// SIMATIC S7-200 project (STEP 7-Micro/WIN), CPU 226 REL 01.23

ORGANIZATION_BLOCK MAIN:OB1
TITLE=
// 项目信息：这个PLC程序控制K650吹瓶机。
// 物理设备包括K650吹瓶机、进料机构、加热区、吹瓶机构、冷却机构、出料机构、传感器和执行器。
// 
// 解析：
// 生产流程从启动按钮按下开始，系统启动后，进料阀门A和进料阀门B打开，将瓶胚送入设备。进料阀门只有在液位传感器未检测到满载、加热区温度传感器显示适宜温度、加热传感器和出料传感器正常、且无急停标志时才会动作，确保进料过程安全无溢料。进料完成后，加热器开始运行，将瓶胚加热至吹瓶所需温度。加热器只有在加热启用标志置位且加热区温度传感器确认温度达标时才会启动，保证瓶胚充分预热。随后，吹瓶机构将加热后的瓶胚吹制成瓶子，在系统确认加热流程结束后启动，避免因加热不足影响质量。
// 吹瓶完成后，冷却器启动，将成型瓶子冷却至适宜温度。冷却器在冷却启用标志置位时启动，确保瓶子冷却均匀、不变形。冷却结束后，出料阀门打开，将成品瓶送出生产线。出料阀门需在出料启用标志置位且出料传感器确认瓶子就位时才会动作，保证出料过程顺畅无堵塞。整个过程中，电机组驱动各环节，确保生产连续性。为保障安全，当急停按钮或急停信号触发时，系统暂停，所有设备停止运行，避免事故发生。
BEGIN
Network 1 // 网络标题
// 网络注释
LDN    V104.1
=      M1.1
?000
Network 2
LD     V600.5
JMP    3
Network 3
LD     I0.5
TON    T180, +2
Network 4
LD     V103.0
A      I3.2
A      I1.2
A      I0.6
A      I1.4
A      I1.1
AN     M1.1
AN     I3.0
AN     I3.1
AN     I3.5
AN     I3.4
AN     T180
LPS
=      M29.0
AN     M1.5
AN     I0.0
AN     M22.1
=      M1.4
LRD
LD     I0.0
O      M1.5
ALD
AN     M22.1
=      M1.5
LPP
LD     I2.5
O      M22.1
ALD
=      M22.1
Network 5
LD     M29.0
CALL   SBR_8:SBR8
Network 6
LD     M29.0
=      Q0.0
Network 7
LD     I0.4
TON    T181, +2
Network 8
LD     V103.0
A      I3.3
A      I0.6
A      I1.4
A      I1.1
AN     M1.1
AN     I3.0
AN     I3.1
AN     I3.5
AN     I3.4
AN     T181
LPS
=      M29.1
AN     M1.7
AN     I0.1
AN     M22.0
=      M1.6
LRD
LD     I0.1
O      M1.7
ALD
AN     M22.0
=      M1.7
LPP
LD     I2.6
O      M22.0
ALD
=      M22.0
Network 9
LD     M29.1
CALL   SBR_1:SBR1
Network 10
LD     M29.1
=      Q0.1
Network 11
LD     V103.0
A      I3.0
A      I1.4
AN     M1.1
AN     I3.2
AN     I3.3
AN     I3.5
AN     I3.4
LDN    I0.7
O      M29.2
ALD
LPS
AN     T214
=      M29.2
LRD
AN     M29.3
AN     M15.1
=      M2.1
LRD
AN     M2.1
TON    T34, +50
LRD
LD     M2.1
O      Q2.2
ALD
AN     T34
AN     M15.1
=      Q2.2
LRD
LD     I2.1
O      M29.3
ALD
AN     M15.1
=      M29.3
LPP
LD     I0.7
O      M15.1
ALD
LPS
AN     T214
=      M15.1
LPP
TON    T214, +5
Network 12
LD     M29.2
CALL   SBR_2:SBR2
Network 13
LD     M29.2
AN     Q0.0
=      Q0.2
Network 14
LD     V103.0
A      I3.1
A      I1.4
AN     M1.1
AN     I3.2
AN     I3.3
AN     I3.5
AN     I0.6
AN     I3.4
LPS
=      M2.3
A      I0.7
AN     M15.3
AN     M15.4
=      M15.2
LRD
AN     I0.7
AN     M15.4
AN     M24.5
=      M15.3
LPP
LD     M24.5
O      M15.4
ALD
=      M15.4
Network 15
LD     M2.3
CALL   SBR_2:SBR2
Network 16
LD     M2.3
=      Q0.3
Network 17
LD     V103.0
A      I3.5
A      I1.4
AN     M1.1
AN     I3.2
AN     I3.3
AN     I3.1
AN     I3.0
AN     I1.0
LPS
=      M29.4
AN     M29.5
AN     I2.3
=      M2.5
LPP
LD     I2.3
O      M29.5
ALD
=      M29.5
Network 18
LD     M29.4
CALL   SBR_3:SBR3
Network 19
LD     M29.4
=      Q1.0
Network 20
LD     V103.0
A      I3.4
A      I1.4
AN     M1.1
AN     I3.2
AN     I3.3
AN     I3.0
AN     I3.1
AN     I1.1
=      M2.7
MOVW   VW452, VW180
MOVW   VW454, VW182
Network 21
LD     M2.7
=      Q1.1
Network 22
LD     V103.0
A      V101.5
A      I1.4
AN     M1.1
=      Q1.2
Network 23
LD     V101.4
A      I1.4
AN     M1.1
=      Q1.3
Network 24
LD     I1.3
TON    T182, +2
Network 25
LD     I3.2
A      V103.1
A      I0.4
A      I1.5
A      I1.4
A      I2.0
AN     M1.1
AN     I3.0
AN     I3.1
AN     I3.4
AN     I3.5
AN     T182
LPS
=      M30.3
AN     M3.2
AN     I0.2
AN     M22.2
=      M3.1
LRD
LD     I0.2
O      M3.2
ALD
AN     M22.2
=      M3.2
LPP
LD     I2.7
O      M22.2
ALD
=      M22.2
Network 26
LD     M30.3
CALL   SBR_4:SBR4
Network 27
LD     M30.3
=      Q1.4
Network 28
LD     I1.2
TON    T183, +2
Network 29
LD     I3.3
A      V103.1
A      I1.5
A      I1.4
A      I2.0
AN     M1.1
AN     I3.0
AN     I3.1
AN     I3.4
AN     I3.5
AN     T183
LPS
=      M30.4
AN     M3.5
AN     I0.3
AN     M22.3
=      M3.4
LRD
LD     I0.3
O      M3.5
ALD
AN     M22.3
=      M3.5
LPP
LD     I3.6
O      M22.3
ALD
=      M22.3
Network 30
LD     M30.4
CALL   SBR_5:SBR5
Network 31
LD     M30.4
=      Q1.5
Network 32
LD     I3.0
A      V103.1
A      I1.4
AN     M1.1
AN     I3.2
AN     I3.3
AN     I3.5
AN     I3.4
LDN    I1.6
O      M29.6
ALD
LPS
AN     T213
=      M29.6
LRD
AN     M29.7
AN     M15.0
=      M3.7
LRD
AN     M3.7
TON    T35, +50
LRD
LD     M3.7
O      Q2.3
ALD
AN     T35
AN     M15.0
=      Q2.3
LRD
LD     I2.2
O      M29.7
ALD
AN     M15.0
=      M29.7
LPP
LD     I1.6
O      M15.0
ALD
LPS
AN     T213
=      M15.0
LPP
TON    T213, +5
Network 33
LD     M29.6
CALL   SBR_2:SBR2
Network 34
LD     M29.6
AN     Q1.4
=      Q1.6
Network 35
LD     I3.1
A      V103.1
A      I1.4
AN     M1.1
AN     I3.2
AN     I3.3
AN     I3.4
AN     I1.5
AN     I3.5
LPS
=      M4.1
A      I1.6
AN     M15.7
AN     M15.6
=      M15.5
LRD
AN     I1.6
AN     M15.7
AN     M24.5
=      M15.6
LPP
LD     M24.5
O      M15.7
ALD
=      M15.7
Network 36
LD     M4.1
CALL   SBR_2:SBR2
Network 37
LD     M4.1
=      Q2.0
Network 38
LD     I3.5
A      V103.1
A      I1.4
AN     M1.1
AN     I3.2
AN     I3.3
AN     I3.1
AN     I3.0
AN     I1.7
LPS
=      M30.0
AN     M30.1
AN     I2.4
=      M4.3
LPP
LD     I2.4
O      M30.1
ALD
=      M30.1
Network 39
LD     M30.0
CALL   SBR_3:SBR3
Network 40
LD     M30.0
=      Q0.4
Network 41
LD     I3.4
A      V103.1
A      I1.4
AN     M1.1
AN     I3.2
AN     I3.3
AN     I3.0
AN     I3.1
AN     I3.1
AN     I2.0
=      M4.5
MOVW   VW452, VW180
MOVW   VW454, VW182
Network 42
LD     M4.5
=      Q0.5
Network 43
LD     V101.5
A      V103.1
A      I1.4
AN     M1.1
=      Q0.6
Network 44
LD     M4.5
O      M4.3
O      M15.5
O      M15.6
O      M3.7
O      M3.4
O      M3.1
O      M2.7
O      M2.5
O      M15.3
O      M15.2
O      M1.6
O      M2.1
O      M1.4
=      Q1.7
Network 45
LD     M1.1
=      V600.5
Network 46
LD     V104.1
O      SM0.1
O      V100.2
R      M10.0, 8
R      M11.0, 2
R      M12.0, 8
R      M13.0, 2
Network 47
LBL    3
Network 48
LDN    V600.5
JMP    1
Network 49
LD     M10.0
O      M10.1
O      M10.2
O      M10.3
=      M20.0
Network 50
LD     M12.0
O      M12.1
O      M12.2
O      M12.3
=      M20.1
Network 51
LDN    M5.6
ON     M5.1
A      M5.2
AN     V104.1
EU
=      M4.7
Network 52
LDN    M5.7
ON     M20.5
A      M5.3
AN     V104.1
EU
=      M5.0
Network 53
LD     M4.7
S      M5.1, 1
Network 54
LD     M5.0
S      M20.5, 1
Network 55
LD     M10.0
A      V100.6
S      M25.2, 1
Network 56
LD     M12.0
A      V100.5
S      M25.3, 1
Network 57
LD     V100.2
O      SM0.1
O      M17.7
LD     V100.3
O      V100.4
ED
OLD
R      M25.2, 2
Network 58
LD     V100.1
S      M7.0, 1
Network 59
LD     SM0.0
MOVW   VW204, VW3800
/I     +2, VW3800
MOVW   VW3800, VW3900
+I     +30, VW3900
Network 60
LD     M7.0
TON    T44, VW3900
Network 61
LD     M10.0
O      SM0.1
O      M27.0
R      M7.0, 1
Network 62
LD     V100.6
AN     M25.2
O      V100.4
AN     M20.1
LD     V100.6
O      V100.4
AN     V100.5
A      V100.1
LD     V100.6
A      V100.5
A      T44
OLD
ALD
LD     T97
A      M7.6
AN     M25.2
OLD
A      M1.1
=      M5.2
Network 63
LD     V100.5
AN     M25.3
O      V100.3
AN     M20.0
A      V100.1
LD     T99
A      M7.6
AN     M25.3
OLD
A      M1.1
=      M5.3
Network 64
LD     V100.1
R      V100.2, 1
Network 65
LD     M4.7
O      M5.0
R      V100.1, 1
Network 66
LD     V100.5
AN     V100.6
LD     V100.6
AN     V100.5
OLD
O      V100.4
O      V100.3
S      M6.0, 1
Network 67
LDN    V100.6
AN     V100.5
O      M20.3
R      M6.2, 1
R      M5.1, 1
R      M20.5, 1
A      Q0.6
A      Q1.2
R      M6.0, 1
Network 68
LDN    V100.6
ON     V100.5
A      M1.1
R      M6.1, 1
Network 69
LD     M5.6
A      M1.1
A      V100.5
TON    T99, VW1316
Network 70
LD     T99
S      V2100.0, 1
Network 71
LD     M12.0
R      V2100.0, 1
Network 72
LD     M12.0
O      V104.1
O      M20.4
O      V100.2
O      M27.0
R      M5.6, 1
Network 73
LD     M1.1
EU
=      M20.4
Network 74
LD     V100.5
A      M10.0
S      M5.6, 1
Network 75
LD     M5.7
A      M1.1
A      V100.6
TON    T97, VW1316
Network 76
LD     T97
S      V2100.1, 1
Network 77
LD     M10.0
R      V2100.1, 1
Network 78
LD     M10.0
O      V104.1
O      M20.3
O      V100.2
O      M27.0
R      M5.7, 1
Network 79
LD     M1.1
EU
=      M20.3
Network 80
LD     V100.6
A      M12.0
S      M5.7, 1
Network 81
LD     V100.6
A      V100.5
S      M6.1, 1
S      M6.2, 1
=      M7.6
Network 82
LD     V100.3
O      V100.2
R      M13.3, 1
Network 83
LD     V100.4
O      V100.2
R      M11.3, 1
Network 84
LDN    M6.5
=      M6.3
Network 85
LD     SM0.1
O      M11.1
O      V100.2
O      V104.1
O      M27.0
R      M6.3, 1
R      M6.5, 1
Network 86
LDN    V100.5
S      M25.0, 1
Network 87
LD     V100.5
A      M10.0
R      M25.0, 1
Network 88
LD     M4.7
A      I0.4
A      I1.2
A      M6.3
LD     M10.0
A      I1.3
OLD
LD     M10.1
A      T139
A      I1.6
OLD
LD     T49
O      T119
O      T120
A      M10.2
AN     V108.5
OLD
LD     M10.3
A      I1.2
LD     M10.4
A      T52
A      I1.7
OLD
LD     M10.5
A      T198
OLD
LD     M10.6
A      T53
OLD
LD     M10.7
A      T148
A      I1.7
OLD
LD     M11.0
A      I1.5
OLD
LD     V108.5
A      T178
OLD
OLD
LD     I2.0
O      T119
O      T120
A      V108.5
A      M10.2
A      T140
LD     M11.1
AN     V108.5
OLD
A      I2.0
OLD
EU
=      M6.4
Network 89
LD     M10.5
TON    T198, +1
Network 90
LD     M11.1
A      V108.5
TON    T178, +5
Network 91
LD     M10.2
A      V108.5
TON    T140, +1
Network 92
LD     M11.2
=      M20.6
Network 93
LD     M11.2
A      M20.7
AN     V100.2
AN     V100.4
LD     I2.0
AN     V108.5
O      V108.5
ALD
A      I1.2
LD     V2100.1
O      M25.0
ALD
LD     V100.6
A      V100.5
O      V100.6
ALD
O      M6.4
A      M1.1
EU
SHRB   M6.3, M10.0, +16
Network 94
LD     M20.6
=      M20.7
Network 95
LD     M10.0
TON    T47, VW950
Network 96
LD     I1.3
TON    T184, +2
Network 97
LD     M10.0
A      T47
LD     M31.5
AN     T184
OLD
A      I1.5
A      I1.4
A      I0.4
LD     I2.0
AN     V108.5
O      V108.5
ALD
A      M1.1
LPS
S      M6.5, 1
=      M31.5
LD     I1.2
O      M6.6
ALD
AN     M6.7
AN     M23.2
=      M6.6
LRD
LD     I0.2
O      M6.7
ALD
AN     M23.2
=      M6.7
LPP
LD     I2.7
O      M23.2
ALD
=      M23.2
Network 98
LD     M31.5
CALL   SBR_4:SBR4
Network 99
LDN    M31.5
TON    T48, VW952
Network 100
LD     M10.1
A      T48
A      I1.4
A      M1.1
A      I1.3
LPS
AN     T139
=      M30.5
LRD
LD     I1.5
O      M30.6
ALD
AN     M8.1
AN     M14.0
=      M30.6
LRD
AN     M30.6
TON    T35, +50
LRD
LD     M30.6
O      Q2.3
ALD
AN     T35
AN     M14.0
=      Q2.3
LRD
LD     I2.2
O      M8.1
ALD
AN     M14.0
=      M8.1
LPP
LD     I1.6
O      M14.0
ALD
LPS
AN     T139
=      M14.0
LPP
TON    T139, +2
Network 101
LD     M30.5
CALL   SBR_2:SBR2
Network 102
LDN    M30.5
TON    T109, VW908
Network 103
LD     M10.1
EU
S      V200.1, 1
Network 104
LD     T199
O      SM0.1
O      M27.0
R      V200.1, 1
Network 105
LD     V200.1
=      M19.6
TON    T100, VW62
Network 106
LD     M10.3
TON    T50, VW956
Network 107
LD     I1.2
TON    T185, +2
Network 108
LD     T50
A      M10.3
LD     M31.6
AN     T185
OLD
A      I2.0
A      I1.4
A      I1.6
A      M1.1
O      M27.5
LPS
=      M31.6
LD     I1.3
O      M27.5
O      M8.4
ALD
AN     M8.5
AN     M23.3
=      M8.4
LRD
LD     I0.3
O      M8.5
ALD
AN     M23.3
=      M8.5
LPP
LD     I3.6
O      M23.3
ALD
=      M23.3
Network 109
LD     M31.6
CALL   SBR_5:SBR5
Network 110
LDN    M31.6
TON    T51, VW958
Network 111
LD     M10.4
A      T51
O      M31.7
A      I1.4
A      M1.1
A      I1.2
LPS
AN     T133
=      M31.7
LRD
AN     M31.0
AN     I2.4
AN     M24.6
AN     I1.7
=      M8.7
LRD
LD     I2.4
O      M31.0
ALD
AN     I1.7
AN     M24.6
=      M31.0
LPP
A      I1.7
LPS
AN     T133
=      M24.6
LPP
TON    T133, VW978
Network 112
LD     M10.7
AN     I1.7
=      M26.3
Network 113
LD     M31.7
O      M26.3
CALL   SBR_3:SBR3
Network 114
LD     M10.4
TON    T166, VW960
Network 115
LD     M10.4
A      T166
A      M1.1
A      I1.4
=      Q0.6
TON    T52, VW204
Network 116
LD     M12.5
A      V100.5
A      V100.6
O      V100.6
O      V100.3
O      V100.5
O      V100.4
A      M1.1
A      M10.6
TON    T53, VW210
=      V600.1
Network 117
LD     M11.0
TON    T55, VW966
Network 118
LD     M10.7
TON    T148, +1
Network 119
LD     T55
A      M11.0
O      M27.3
AN     I1.5
LPS
A      M1.1
=      M9.1
LPP
LD     I1.6
ON     I1.6
ALD
=      M14.5
Network 120
LD     M9.1
CALL   SBR_2:SBR2
Network 121
LD     M9.1
A      M1.1
O      M27.3
AN     I1.5
LD     Q0.0
A      V100.5
AN     Q0.6
AN     V100.4
AN     V100.6
OLD
=      Q2.0
Network 122
LD     M11.1
TON    T58, VW964
Network 123
LD     V600.1
TON    T54, VW980
Network 124
LD     M11.1
A      T58
A      I1.4
AN     V108.5
A      I1.5
A      M1.1
LD     M10.2
A      V108.5
OLD
LDN    T54
A      V600.1
OLD
O      M27.4
AN     I2.0
=      M8.2
MOVW   VW452, VW180
MOVW   VW454, VW182
Network 125
LD     M8.2
O      M27.4
A      M1.1
=      Q0.5
Network 126
LDN    M9.6
A      M1.1
=      M9.2
Network 127
LD     SM0.1
O      M13.1
O      V100.2
O      V104.1
O      M17.7
R      M9.2, 1
R      M9.6, 1
Network 128
LDN    V100.6
S      M25.1, 1
Network 129
LD     V100.6
A      M12.0
R      M25.1, 1
Network 130
LD     M5.0
A      I1.2
A      I0.4
A      M9.2
LD     M12.0
A      I0.5
OLD
LD     M12.1
A      I0.7
A      T131
OLD
LD     T39
O      T119
O      T120
A      M12.2
AN     V108.5
OLD
LD     M12.3
A      I0.4
LD     M12.4
A      T42
A      I1.0
OLD
LD     M12.5
A      T159
OLD
LD     M12.6
A      T43
OLD
LD     M12.7
A      T149
A      I1.0
OLD
LD     M13.0
A      I0.6
OLD
LD     T143
A      V108.5
OLD
OLD
LD     I1.1
O      T39
O      T119
A      T141
A      M12.2
A      V108.5
LD     M13.1
AN     V108.5
OLD
A      I1.1
OLD
EU
=      M9.3
Network 131
LD     M13.1
A      V108.5
TON    T143, +5
Network 132
LD     M12.2
A      V108.5
TON    T141, +1
Network 133
LD     M12.5
TON    T159, +1
Network 134
LD     M12.7
TON    T149, +1
Network 135
LD     M13.2
=      M21.0
Network 136
LD     M13.2
A      M21.1
LD     V2100.0
O      M25.1
ALD
AN     V100.2
AN     V100.3
LD     I1.1
AN     V108.5
O      V108.5
ALD
A      I0.4
LD     V100.5
A      V100.6
O      V100.5
ALD
O      M9.3
A      M1.1
EU
SHRB   M9.2, M12.0, +16
Network 137
LD     M21.0
=      M21.1
Network 138
LD     M12.0
TON    T37, VW900
Network 139
LD     I0.5
TON    T186, +2
Network 140
LD     I1.1
AN     V108.5
O      V108.5
LD     M12.0
A      T37
LD     M28.0
AN     T186
OLD
ALD
A      I0.6
A      I1.4
A      M1.1
A      I1.2
LPS
=      M28.0
LD     I0.4
O      M9.4
ALD
AN     M9.5
AN     I0.0
AN     M23.0
=      M9.4
LRD
LD     I0.0
O      M9.5
ALD
AN     M23.0
=      M9.5
LRD
S      M9.6, 1
LPP
LD     I2.5
O      M23.0
ALD
=      M23.0
Network 141
LD     M28.0
CALL   SBR_8:SBR8
Network 142
LDN    M28.0
TON    T38, VW904
Network 143
LD     M12.1
A      T38
A      I1.4
A      M1.1
A      I0.5
LPS
AN     T131
=      M31.1
LRD
LD     I0.6
O      M31.2
ALD
AN     M17.0
AN     M14.1
=      M31.2
LRD
AN     M31.2
TON    T36, +50
LRD
LD     M31.2
O      Q2.2
ALD
AN     T36
AN     M14.1
=      Q2.2
LRD
LD     I2.1
O      M17.0
ALD
AN     M14.1
=      M17.0
LPP
LD     I0.7
O      M14.1
ALD
LPS
AN     T131
=      M14.1
LPP
TON    T131, +2
Network 144
LD     M31.1
CALL   SBR_2:SBR2
Network 145
LDN    M31.1
TON    T114, VW908
Network 146
LD     M12.1
EU
S      V200.0, 1
Network 147
LD     T199
O      M27.0
O      SM0.1
R      V200.0, 1
Network 148
LD     V200.0
=      M19.7
TON    T98, VW60
Network 149
LD     T98
O      T100
LD     Q2.1
AN     T199
OLD
=      Q2.1
Network 150
LD     Q2.1
TON    T199, VW236
Network 151
LD     M12.3
TON    T40, VW912
Network 152
LD     I0.4
TON    T187, +2
Network 153
LD     M12.3
A      T40
LD     M28.1
AN     T187
OLD
A      I1.1
A      I1.4
A      M1.1
A      I0.7
O      M27.2
LPS
=      M28.1
LD     I0.5
O      M27.2
O      M17.3
ALD
AN     M17.4
AN     I0.1
AN     M23.1
=      M17.3
LRD
LD     I0.1
O      M17.4
ALD
AN     M23.1
=      M17.4
LPP
LD     I2.6
O      M23.1
ALD
=      M23.1
Network 154
LD     M28.1
CALL   SBR_1:SBR1
Network 155
LDN    M28.1
TON    T41, VW902
Network 156
LD     M12.4
A      T41
O      M28.2
A      I1.4
A      M1.1
A      I0.4
LPS
AN     T132
=      M28.2
LRD
AN     M31.4
AN     I2.3
AN     M24.7
AN     I1.0
=      M17.6
LRD
LD     I2.3
O      M31.4
ALD
AN     I1.0
AN     M24.7
=      M31.4
LPP
A      I1.0
LPS
AN     T132
=      M24.7
LPP
TON    T132, VW978
Network 157
LD     M12.7
AN     I1.0
=      M26.4
Network 158
LD     M28.2
O      M26.4
CALL   SBR_3:SBR3
Network 159
LD     M12.4
TON    T144, VW906
Network 160
LD     M12.4
A      T144
A      M1.1
A      I1.4
=      Q1.2
TON    T42, VW204
Network 161
LD     M10.5
A      V100.5
A      V100.6
O      V100.3
O      V100.4
O      V100.6
O      V100.5
A      M1.1
A      M12.6
TON    T43, VW210
=      V600.0
Network 162
LD     M13.0
TON    T45, VW910
Network 163
LD     T45
A      M13.0
O      M27.0
AN     I0.6
LPS
A      M1.1
=      M16.0
LPP
LD     I0.7
ON     I0.7
ALD
=      M14.2
Network 164
LD     M16.0
O      V3000.3
CALL   SBR_2:SBR2
Network 165
LDN    M16.0
TON    T46, VW914
Network 166
LD     V600.0
TON    T57, VW980
Network 167
LD     M13.1
A      T46
A      I1.4
AN     V108.5
A      I0.6
LD     M12.2
A      V108.5
OLD
LD     V600.0
AN     T57
OLD
O      M27.1
A      M1.1
AN     I1.1
=      M17.1
MOVW   VW452, VW180
MOVW   VW454, VW182
Network 168
LD     M17.1
O      M27.1
A      M1.1
=      Q1.1
Network 169
LD     M16.0
AN     Q1.4
O      M27.0
A      M1.1
AN     I0.6
LD     Q1.4
A      V100.6
AN     Q1.2
AN     V100.5
AN     V100.3
OLD
=      Q0.3
Network 170
LD     M28.0
A      M1.1
=      Q0.0
Network 171
LD     M31.1
O      M24.7
A      M1.1
=      Q0.2
Network 172
LD     M28.1
A      M1.1
O      M27.2
=      Q0.1
Network 173
LD     M31.5
A      M1.1
=      Q1.4
Network 174
LD     M30.5
O      M24.6
A      M1.1
=      Q1.6
Network 175
LD     M31.6
A      M1.1
O      M27.5
=      Q1.5
Network 176
LD     M31.0
O      M8.7
O      M31.7
O      M26.3
A      M1.1
=      Q0.4
Network 177
LD     M17.6
O      M31.4
O      M28.2
O      M26.4
A      M1.1
=      Q1.0
Network 178
LD     M17.0
O      M8.1
O      M17.1
O      M14.3
O      M14.2
O      M17.6
O      M17.3
O      M31.2
O      M8.2
O      M14.6
O      M14.5
O      M8.7
O      M8.4
O      M30.6
O      M6.6
O      M9.4
=      Q1.7
Network 179
LD     V108.0
A      M1.1
EU
=      M17.7
Network 180
LD     M27.0
O      V108.0
R      M10.0, 8
R      M11.0, 2
R      M12.0, 8
R      M13.0, 2
Network 181
LD     M27.0
R      V108.0, 1
Network 182
LD     M17.7
A      M1.1
AN     M7.5
LD     M27.0
A      T160
A      I0.6
OLD
LD     M27.1
A      T161
A      I1.1
OLD
LD     M27.2
A      T162
A      I0.4
OLD
LD     M27.3
A      T163
A      I1.5
OLD
LD     M27.4
A      T164
A      I2.0
OLD
LD     M27.5
A      T165
A      I1.2
OLD
EU
=      M7.4
Network 183
LD     M27.0
O      M27.1
O      M27.2
O      M27.3
O      M27.4
O      M27.5
=      M7.5
Network 184
LD     M27.0
TON    T160, +5
Network 185
LD     M27.1
TON    T161, +5
Network 186
LD     M27.2
TON    T162, +5
Network 187
LD     M27.3
TON    T163, +5
Network 188
LD     M27.4
TON    T164, +5
Network 189
LD     M27.5
TON    T165, +5
Network 190
LD     M7.4
EU
SHRB   M17.7, M27.0, +6
Network 191
LD     I2.0
A      I1.1
A      I0.4
A      I0.6
A      I1.5
A      I1.2
O      SM0.1
O      V100.1
R      M27.0, 6
R      V108.0, 1
Network 192
LDN    V102.0
JMP    0
Network 193
LD     M10.2
O      M12.2
EU
S      M0.3, 1
Network 194
LD     M0.3
TON    T190, VW908
Network 195
LD     T49
R      M0.3, 1
Network 196
LD     T190
A      M1.1
LD     Q1.3
AN     T49
OLD
=      Q1.3
TON    T49, VW216
TON    T39, VW216
Network 197
LD     T49
S      M16.1, 1
Network 198
LD     M16.1
AN     T103
=      M16.2
TON    T103, VW216
Network 199
LD     T103
R      M16.1, 1
Network 200
LBL    0
Network 201
LD     V102.0
JMP    2
Network 202
LD     M10.2
O      M12.2
S      M0.4, 1
Network 203
LD     M0.4
TON    T196, VW908
Network 204
LD     T119
O      T120
R      M0.4, 1
Network 205
LD     T196
AN     T119
A      M1.1
A      M16.4
R      M16.2, 1
S      Q1.3, 1
TON    T119, +1
Network 206
LD     T196
AN     T120
A      M16.3
O      SM0.1
R      Q1.3, 1
S      M16.2, 1
TON    T120, +1
Network 207
LD     Q1.3
A      M1.1
TON    T105, +10
Network 208
LDN    Q1.3
A      M1.1
TON    T106, +10
Network 209
LD     T105
R      M16.4, 1
S      M16.3, 1
Network 210
LD     T106
O      SM0.1
R      M16.3, 1
S      M16.4, 1
Network 211
LBL    2
Network 212
LD     M12.4
O      M10.4
A      M6.0
LD     M6.3
AN     M16.5
OLD
LD     M12.4
O      M10.4
A      M6.1
OLD
AN     T212
A      M1.1
TON    T212, +2
Network 213
LD     SM0.1
O      V104.1
O      V100.2
R      M16.5, 1
Network 214
LD     M10.0
O      M12.0
S      M16.5, 1
Network 215
LD     T212
EU
=      M0.0
Network 216
LD     M1.1
=      V600.5
Network 217
LBL    1
Network 218
LD     SM0.0
CALL   SBR_9:SBR9
Network 219
LD     SM0.0
END
END_ORGANIZATION_BLOCK

SUBROUTINE_BLOCK SBR_57:SBR0
TITLE=子程序注释
VAR_INPUT
setting:INT;	// LW0 
input:WORD;	// LW2 
sh_p:WORD;	// LW4 
x_p:WORD;	// LW6 
temp_sw1:BOOL;	// L8.0 
heat_q:BOOL;	// L8.1 
cool_q:BOOL;	// L8.2 
END_VAR
VAR_IN_OUT
prerent:INT;	// LW9 
END_VAR
VAR_OUTPUT
temp_ok:BOOL;	// L11.0 
sh_a:BOOL;	// L11.1 
x_a:BOOL;	// L11.2 
temp_status:BYTE;	// LB12 
END_VAR
BEGIN
Network 1 // 网络标题
// 网络注释
LD     SM0.0
LPS
MOVW   #input:LW2, #prerent:LW9
/I     +10, #prerent:LW9
MOVW   #prerent:LW9, LW14
AENO
+I     #x_p:LW6, LW14
AENO
AW>=   LW14, #setting:LW0
=      #temp_ok:L11.0
LRD
MOVW   #setting:LW0, LW14
AENO
+I     #sh_p:LW4, LW14
AENO
AW>    #prerent:LW9, LW14
A      #temp_sw1:L8.0
AW<>   #setting:LW0, +0
=      #sh_a:L11.1
LPP
MOVW   #setting:LW0, LW14
AENO
-I     #x_p:LW6, LW14
AENO
AW<    #prerent:LW9, LW14
A      #temp_sw1:L8.0
AW<>   #setting:LW0, +0
=      #x_a:L11.2
Network 2
LDN    #cool_q:L8.2
AN     #heat_q:L8.1
MOVB   0, #temp_status:LB12
Network 3
LDN    #cool_q:L8.2
A      #heat_q:L8.1
MOVB   1, #temp_status:LB12
Network 4
LD     #cool_q:L8.2
AN     #heat_q:L8.1
MOVB   1, #temp_status:LB12
END_SUBROUTINE_BLOCK

SUBROUTINE_BLOCK SBR_1:SBR1
TITLE=
BEGIN
Network 1
LD     M1.6
O      M17.3
MOVW   VW408, VW180
MOVW   VW410, VW182
Network 2
LD     M1.7
O      M17.4
MOVW   VW412, VW180
AENO
MOVW   VW414, VW182
Network 3
LD     M22.0
O      M23.1
MOVW   VW604, VW180
AENO
MOVW   VW606, VW182
AENO
CRET
END_SUBROUTINE_BLOCK

SUBROUTINE_BLOCK SBR_2:SBR2
TITLE=
BEGIN
Network 1
LD     M2.1
O      M31.2
O      M30.6
O      M3.7
MOVW   VW432, VW180
MOVW   VW434, VW182
Network 2
LD     M29.3
O      M17.0
O      M8.1
O      M29.7
MOVW   VW436, VW180
AENO
MOVW   VW438, VW182
Network 3
LD     M14.1
O      M15.1
O      M15.0
O      M14.0
MOVW   VW440, VW180
AENO
MOVW   VW442, VW182
Network 4
LD     M14.5
O      M14.6
O      M15.5
O      M15.6
O      M14.7
O      M15.7
O      M14.2
O      M14.3
O      M15.2
O      M15.3
O      M14.4
O      M15.4
MOVW   VW970, VW180
AENO
MOVW   VW972, VW182
AENO
CRET
END_SUBROUTINE_BLOCK

SUBROUTINE_BLOCK SBR_3:SBR3
TITLE=
BEGIN
Network 1
LD     M2.5
O      M4.3
O      M17.6
O      M8.7
MOVW   VW444, VW180
MOVW   VW446, VW182
Network 2
LD     M29.5
O      M30.1
O      M31.4
O      M31.0
O      M26.3
O      M26.4
MOVW   VW448, VW180
AENO
MOVW   VW450, VW182
Network 3
LD     M24.6
O      M24.7
MOVW   VW440, VW180
AENO
MOVW   VW442, VW182
AENO
CRET
END_SUBROUTINE_BLOCK

SUBROUTINE_BLOCK SBR_4:SBR4
TITLE=
BEGIN
Network 1
LD     M3.1
O      M6.6
MOVW   VW416, VW180
MOVW   VW418, VW182
Network 2
LD     M3.2
O      M6.7
MOVW   VW420, VW180
AENO
MOVW   VW422, VW182
Network 3
LD     M22.2
O      M23.2
MOVW   VW608, VW180
AENO
MOVW   VW610, VW182
AENO
CRET
END_SUBROUTINE_BLOCK

SUBROUTINE_BLOCK SBR_5:SBR5
TITLE=
BEGIN
Network 1
LD     M3.4
O      M8.4
MOVW   VW424, VW180
MOVW   VW426, VW182
Network 2
LD     M3.5
O      M8.5
MOVW   VW428, VW180
AENO
MOVW   VW430, VW182
Network 3
LD     M22.3
O      M23.3
MOVW   VW612, VW180
AENO
MOVW   VW618, VW182
AENO
CRET
END_SUBROUTINE_BLOCK

SUBROUTINE_BLOCK SBR_8:SBR8
TITLE=
BEGIN
Network 1
LD     M1.4
O      M9.4
MOVW   VW400, VW180
MOVW   VW402, VW182
Network 2
LD     M1.5
O      M9.5
MOVW   VW404, VW180
AENO
MOVW   VW406, VW182
Network 3
LD     M22.1
O      M23.0
MOVW   VW616, VW180
AENO
MOVW   VW602, VW182
AENO
CRET
END_SUBROUTINE_BLOCK

SUBROUTINE_BLOCK SBR_9:SBR9
TITLE=
BEGIN
Network 1
LD     SM0.1
R      V4100.6, 1
S      V4100.5, 1
Network 2
LD     T241
S      V4100.5, 1
R      V4100.6, 1
Network 3
LD     V4100.5
TON    T240, +50
Network 4
LD     T240
R      V4100.5, 1
S      V4100.6, 1
Network 5
LD     V4100.6
TON    T241, +50
Network 6
LD     SM0.0
CALL   SBR_57:SBR0, VW220, AIW0, VW72, VW74, V105.1, Q2.4, Q3.0, VW260, V3200.0, V3200.1, V3200.2, VB1040
Network 7
LDN    V105.1
JMP    5
Network 8
LD     SM0.0
LPS
MOVW   VW260, LW0
AENO
+I     +10, LW0
AENO
AW<    LW0, VW220
JMP    1
LRD
AW<=   VW260, VW220
JMP    2
LRD
MOVW   VW260, LW0
AENO
-I     +5, LW0
AENO
AW>=   LW0, VW220
JMP    3
LRD
MOVW   VW260, LW0
AENO
-I     +10, LW0
AENO
AW>=   LW0, VW220
JMP    4
LPP
JMP    6
Network 9
LBL    1
Network 10
LD     SM0.0
S      Q2.4, 1
R      Q3.0, 1
JMP    6
Network 11
LBL    2
Network 12
LD     SM0.0
LPS
MOVW   VW220, LW0
AENO
-I     VW260, LW0
AENO
MOVW   LW0, LW1
AENO
*I     +10, LW1
AENO
MOVW   LW1, VW1400
+I     +10, VW1400
LRD
A      V4100.5
S      Q2.4, 1
LPP
R      Q3.0, 1
Network 13
LD     Q2.4
TON    T254, VW1400
Network 14
LD     T254
R      Q2.4, 1
Network 15
LD     SM0.0
JMP    6
Network 16
LBL    3
Network 17
LD     SM0.0
LPS
MOVW   VW260, LW0
AENO
-I     VW220, LW0
AENO
MOVW   LW0, LW1
AENO
*I     +10, LW1
AENO
MOVW   LW1, VW1402
+I     +10, VW1402
LRD
A      V4100.5
A      V106.1
S      Q3.0, 1
LPP
R      Q2.4, 1
Network 18
LD     Q3.0
TON    T253, VW1402
Network 19
LD     T253
O      V106.2
R      Q3.0, 1
Network 20
LD     SM0.0
JMP    6
Network 21
LBL    4
Network 22
LDW<=  VW260, VW220
R      Q3.1, 1
Network 23
LD     SM0.0
S      Q3.0, 1
R      Q2.4, 1
JMP    6
Network 24
LBL    5
Network 25
LDN    V105.1
R      Q2.4, 1
R      Q3.0, 1
Network 26
LBL    6
Network 27
LD     SM0.0
CALL   SBR_57:SBR0, VW222, AIW2, VW72, VW74, V105.2, Q2.5, Q3.1, VW262, V3200.3, V3200.4, V3200.5, VB1041
Network 28
LDN    V105.2
JMP    11
Network 29
LD     SM0.0
LPS
MOVW   VW262, LW0
AENO
+I     +10, LW0
AENO
AW<    LW0, VW222
JMP    7
LRD
AW<=   VW262, VW222
JMP    8
LRD
MOVW   VW262, LW0
AENO
-I     +5, LW0
AENO
AW>    LW0, VW222
JMP    9
LRD
MOVW   VW262, LW0
AENO
-I     +2, LW0
AENO
AW>=   LW0, VW222
JMP    10
LPP
JMP    12
Network 30
LBL    7
Network 31
LD     SM0.0
S      Q2.5, 1
R      Q3.1, 1
JMP    12
Network 32
LBL    8
Network 33
LD     SM0.0
LPS
MOVW   VW222, LW0
AENO
-I     VW262, LW0
AENO
MOVW   LW0, LW1
AENO
*I     +10, LW1
AENO
MOVW   LW1, VW1404
+I     +10, VW1404
LRD
A      V4100.6
S      Q2.5, 1
LPP
R      Q3.1, 1
Network 34
LD     Q2.5
TON    T252, VW1404
Network 35
LD     T252
R      Q2.5, 1
Network 36
LD     SM0.0
JMP    12
Network 37
LBL    9
Network 38
LD     SM0.0
LPS
MOVW   VW262, LW0
AENO
-I     VW222, LW0
AENO
MOVW   LW0, LW1
AENO
*I     +10, LW1
AENO
MOVW   LW1, VW1406
+I     +10, VW1406
LRD
A      V4100.6
A      V106.4
S      Q3.1, 1
LPP
R      Q2.5, 1
Network 39
LD     Q3.1
TON    T251, VW1406
Network 40
LD     T251
O      V106.5
R      Q3.1, 1
Network 41
LD     SM0.0
JMP    12
Network 42
LBL    10
Network 43
LDW<=  VW262, VW222
R      Q3.1, 1
Network 44
LD     V106.4
A      SM0.0
S      Q3.1, 1
R      Q2.5, 1
JMP    12
Network 45
LBL    11
Network 46
LDN    V105.2
R      Q2.5, 1
R      Q3.1, 1
Network 47
LBL    12
Network 48
LD     SM0.0
CALL   SBR_57:SBR0, VW224, AIW4, VW72, VW74, V105.3, Q2.6, Q3.2, VW264, V3200.6, V3200.7, V3201.0, VB1042
Network 49
LDN    V105.3
JMP    17
Network 50
LD     SM0.0
LPS
MOVW   VW264, LW0
AENO
+I     +10, LW0
AENO
AW<    LW0, VW224
JMP    13
LRD
AW<=   VW264, VW224
JMP    14
LRD
MOVW   VW264, LW0
AENO
-I     +5, LW0
AENO
AW>    LW0, VW224
JMP    15
LRD
MOVW   VW264, LW0
AENO
-I     +10, LW0
AENO
AW>=   LW0, VW224
JMP    16
LPP
JMP    18
Network 51
LBL    13
Network 52
LD     SM0.0
S      Q2.6, 1
R      Q3.2, 1
JMP    18
Network 53
LBL    14
Network 54
LD     SM0.0
LPS
MOVW   VW224, LW0
AENO
-I     VW264, LW0
AENO
MOVW   LW0, LW1
AENO
*I     +10, LW1
AENO
MOVW   LW1, VW1408
+I     +10, VW1408
LRD
A      V4100.5
S      Q2.6, 1
LPP
R      Q3.2, 1
Network 55
LD     Q2.6
TON    T250, VW1408
Network 56
LD     T250
R      Q2.6, 1
Network 57
LD     SM0.0
JMP    18
Network 58
LBL    15
Network 59
LD     SM0.0
LPS
MOVW   VW264, LW0
AENO
-I     VW224, LW0
AENO
MOVW   LW0, LW1
AENO
*I     +10, LW1
AENO
MOVW   LW1, VW1410
+I     +5, VW1410
LRD
A      V4100.5
A      V107.1
S      Q3.2, 1
LPP
R      Q2.6, 1
Network 60
LD     Q3.2
TON    T249, VW1410
Network 61
LD     T249
O      V107.2
R      Q3.2, 1
Network 62
LD     SM0.0
JMP    18
Network 63
LBL    16
Network 64
LDW<=  VW264, VW224
R      Q3.1, 1
Network 65
LD     V107.1
A      SM0.0
S      Q3.2, 1
R      Q2.6, 1
JMP    18
Network 66
LBL    17
Network 67
LDN    V105.3
R      Q2.6, 1
R      Q3.2, 1
Network 68
LBL    18
Network 69
LD     SM0.0
CALL   SBR_57:SBR0, VW226, AIW6, VW72, VW74, V105.4, Q2.7, L4.0, VW266, V3201.1, V3201.2, V3201.3, VB1043
Network 70
LDN    V105.4
JMP    23
Network 71
LD     SM0.0
LPS
MOVW   VW266, LW0
AENO
+I     +2, LW0
AENO
AW<    LW0, VW226
JMP    19
LRD
AW<=   VW266, VW226
JMP    20
LRD
MOVW   VW266, LW0
AENO
-I     +2, LW0
AENO
AW<    LW0, VW226
JMP    21
LRD
MOVW   VW266, LW0
AENO
-I     +2, LW0
AENO
AW>=   LW0, VW226
JMP    22
LPP
JMP    24
Network 72
LBL    19
Network 73
LD     SM0.0
S      Q2.7, 1
R      L4.0, 1
JMP    24
Network 74
LBL    20
Network 75
LD     SM0.0
LPS
MOVW   VW226, LW0
AENO
-I     VW266, LW0
AENO
MOVW   LW0, LW1
AENO
*I     +10, LW1
AENO
MOVW   LW1, VW1412
+I     +10, VW1412
LRD
A      V4100.6
S      Q2.7, 1
LPP
R      L4.0, 1
Network 76
LD     Q2.7
TON    T248, VW1412
Network 77
LD     T248
R      Q2.7, 1
Network 78
LD     SM0.0
JMP    24
Network 79
LBL    21
Network 80
LD     SM0.0
LPS
MOVW   VW266, LW0
AENO
-I     VW226, LW0
AENO
MOVW   LW0, VW1414
+I     +10, VW1414
LRD
A      V4100.6
S      L4.0, 1
LPP
R      Q2.7, 1
Network 81
LD     L4.0
TON    T247, VW1414
Network 82
LD     T247
R      L4.0, 1
Network 83
LD     SM0.0
JMP    24
Network 84
LBL    22
Network 85
LD     SM0.0
R      L4.0, 1
R      Q2.7, 1
JMP    24
Network 86
LBL    23
Network 87
LDN    V105.4
R      Q2.7, 1
R      L4.0, 1
Network 88
LBL    24
Network 89
LD     SM0.0
CALL   SBR_57:SBR0, VW228, AIW8, VW72, VW74, V105.5, Q3.4, L4.0, VW268, V3201.4, V3201.5, V3201.6, VB1044
Network 90
LDN    V105.5
JMP    29
Network 91
LD     SM0.0
LPS
MOVW   VW268, LW0
AENO
+I     +2, LW0
AENO
AW<    LW0, VW228
JMP    25
LRD
AW<=   VW268, VW228
JMP    26
LRD
AW>    VW268, VW228
JMP    28
LPP
JMP    30
Network 92
LBL    25
Network 93
LD     SM0.0
S      Q3.4, 1
JMP    30
Network 94
LBL    26
Network 95
LD     SM0.0
LPS
MOVW   VW228, LW0
AENO
-I     VW268, LW0
AENO
MOVW   LW0, LW1
AENO
*I     +10, LW1
AENO
MOVW   LW1, VW1416
+I     +10, VW1416
LPP
A      V4100.5
S      Q3.4, 1
Network 96
LD     Q3.4
TON    T246, VW1416
Network 97
LD     T246
R      Q3.4, 1
Network 98
LD     SM0.0
JMP    30
Network 99
LBL    28
Network 100
LD     SM0.0
R      Q3.4, 1
JMP    30
Network 101
LBL    29
Network 102
LDN    V105.5
R      Q3.4, 1
Network 103
LBL    30
Network 104
LD     SM0.0
CALL   SBR_57:SBR0, VW230, AIW10, VW72, VW74, V105.6, Q3.5, L4.0, VW270, V3201.7, V3202.0, V3202.1, VB1045
Network 105
LDN    V105.6
JMP    35
Network 106
LD     SM0.0
LPS
MOVW   VW270, LW0
AENO
+I     +2, LW0
AENO
AW<    LW0, VW230
JMP    31
LRD
AW<=   VW270, VW230
JMP    32
LRD
AW>    VW270, VW230
JMP    34
LPP
JMP    36
Network 107
LBL    31
Network 108
LD     SM0.0
S      Q3.5, 1
JMP    36
Network 109
LBL    32
Network 110
LD     SM0.0
LPS
MOVW   VW230, LW0
AENO
-I     VW270, LW0
AENO
MOVW   LW0, LW1
AENO
*I     +10, LW1
AENO
MOVW   LW1, VW1420
+I     +10, VW1420
LPP
A      V4100.6
S      Q3.5, 1
Network 111
LD     Q3.5
TON    T245, VW1420
Network 112
LD     T245
R      Q3.5, 1
Network 113
LD     SM0.0
JMP    36
Network 114
LBL    34
Network 115
LD     SM0.0
R      Q3.5, 1
JMP    36
Network 116
LBL    35
Network 117
LDN    V105.6
R      Q3.5, 1
Network 118
LBL    36
Network 119
LD     SM0.0
CALL   SBR_57:SBR0, VW232, AIW12, VW72, VW74, V105.7, Q3.6, L4.0, VW272, V3202.2, V3202.3, V3202.4, VB1046
Network 120
LDN    V105.7
JMP    41
Network 121
LD     SM0.0
LPS
MOVW   VW272, LW0
AENO
+I     +2, LW0
AENO
AW<    LW0, VW232
JMP    37
LRD
AW<=   VW272, VW232
JMP    38
LRD
AW>    VW272, VW232
JMP    40
LPP
JMP    42
Network 122
LBL    37
Network 123
LD     SM0.0
S      Q3.6, 1
JMP    42
Network 124
LBL    38
Network 125
LD     SM0.0
LPS
MOVW   VW232, LW0
AENO
-I     VW272, LW0
AENO
MOVW   LW0, LW1
AENO
*I     +10, LW1
AENO
MOVW   LW1, VW1424
+I     +10, VW1424
LPP
A      V4100.5
S      Q3.6, 1
Network 126
LD     Q3.6
TON    T244, VW1424
Network 127
LD     T244
R      Q3.6, 1
Network 128
LD     SM0.0
JMP    42
Network 129
LBL    40
Network 130
LD     SM0.0
R      Q3.6, 1
JMP    42
Network 131
LBL    41
Network 132
LDN    V105.7
R      Q3.6, 1
Network 133
LBL    42
Network 134
LD     SM0.0
CALL   SBR_57:SBR0, VW234, AIW14, VW72, VW74, V17.4, Q3.7, L4.0, VW274, V3202.5, V3202.6, V3202.7, VB1047
Network 135
LDN    V17.4
JMP    47
Network 136
LD     SM0.0
LPS
MOVW   VW274, LW0
AENO
+I     +2, LW0
AENO
AW<    LW0, VW234
JMP    43
LRD
AW<=   VW274, VW234
JMP    44
LRD
AW>    VW274, VW234
JMP    46
LPP
JMP    48
Network 137
LBL    43
Network 138
LD     SM0.0
S      Q3.7, 1
JMP    48
Network 139
LBL    44
Network 140
LD     SM0.0
LPS
MOVW   VW234, LW0
AENO
-I     VW274, LW0
AENO
MOVW   LW0, LW1
AENO
*I     +10, LW1
AENO
MOVW   LW1, VW1428
+I     +10, VW1428
LPP
A      V4100.5
S      Q3.7, 1
Network 141
LD     Q3.7
TON    T243, VW1428
Network 142
LD     T243
R      Q3.7, 1
Network 143
LD     SM0.0
JMP    48
Network 144
LBL    46
Network 145
LD     SM0.0
R      Q3.7, 1
JMP    48
Network 146
LBL    47
Network 147
LDN    V17.4
R      Q3.7, 1
Network 148
LBL    48
Network 149
LDN    M29.0
AN     M29.1
AN     M29.2
AN     M2.3
AN     M29.4
=      M18.7
Network 150
LD     M18.7
AN     M2.7
AN     M30.3
AN     M30.4
AN     M24.6
AN     M24.7
=      M18.0
Network 151
LD     M18.0
AN     M29.6
AN     M4.1
AN     M30.0
AN     M26.3
AN     M26.4
=      M19.0
Network 152
LD     M19.0
AN     M4.5
AN     M31.5
AN     M30.5
AN     M8.2
AN     M31.6
=      M18.1
Network 153
LD     M18.1
AN     M31.7
AN     M9.1
AN     M28.0
AN     M14.0
=      M19.1
Network 154
LD     M19.1
AN     M31.1
AN     M17.1
AN     M28.1
AN     M28.2
AN     M16.0
=      M28.7
Network 155
LD     M28.7
O      SM0.1
MOVW   +0, AQW0
MOVW   +0, AQW2
Network 156
LD     M29.0
O      M29.1
O      M29.2
O      M2.3
O      M24.7
O      M24.6
=      M18.5
Network 157
LD     M18.5
O      M29.4
O      M2.7
O      M30.3
O      M30.4
O      M26.3
O      M26.4
=      M18.2
Network 158
LD     M18.2
O      M29.6
O      M4.1
O      M30.0
=      M18.4
Network 159
LD     M18.4
O      M4.5
O      M31.5
O      M30.5
O      M8.2
O      M31.6
=      M18.3
Network 160
LD     M18.3
O      M31.7
O      M9.1
O      M28.0
=      M18.6
Network 161
LD     M18.6
O      M31.1
O      M17.1
O      M28.1
O      M28.2
O      M16.0
=      M28.6
Network 162
LD     M28.6
MOVW   +320, VW806
AENO
*I     VW180, VW806
AENO
MOVW   +320, VW808
AENO
*I     VW182, VW808
AENO
MOVW   VW806, AQW0
AENO
MOVW   VW808, AQW2
Network 163
LD     V104.0
EU
MOVD   +0, VD284
Network 164
LD     Q0.0
O      Q1.4
A      M1.1
EU
INCD   VD284
INCD   VD280
Network 165
LD     M29.0
O      M28.0
=      V301.0
Network 166
LD     M29.1
O      M28.1
=      V301.1
Network 167
LD     M29.2
O      M31.1
=      V301.2
Network 168
LD     M2.3
O      M16.0
=      V301.3
Network 169
LD     M2.7
O      M17.1
=      V301.4
Network 170
LD     M29.4
O      M28.2
=      V301.5
Network 171
LD     Q1.3
=      V301.6
Network 172
LD     Q1.2
=      V301.7
Network 173
LD     V600.0
=      V300.0
Network 174
LD     M30.3
O      M31.5
=      V300.3
Network 175
LD     M30.4
O      M31.6
=      V300.4
Network 176
LD     M29.6
O      M30.5
=      V300.5
Network 177
LD     M4.1
O      M9.1
=      V300.6
Network 178
LD     M4.5
O      M8.2
=      V300.7
Network 179
LD     M30.0
O      M31.7
=      V303.0
Network 180
LD     Q0.6
=      V303.2
Network 181
LD     V600.1
=      V303.3
Network 182
LD     SM0.0
R      V104.0, 1
Network 183
LD     V104.1
R      M27.0, 7
Network 184
LDN    T167
A      M1.2
=      V303.1
Network 185
LD     SM0.1
S      M1.3, 1
Network 186
LD     T167
LPS
AN     M1.3
=      Q3.3
LPP
R      M1.3, 1
Network 187
LDN    T189
AN     M1.2
TON    T167, VW70
Network 188
LD     V105.1
AN     V3200.0
LD     V105.2
AN     V3200.3
OLD
LD     V105.3
AN     V3200.6
OLD
LD     V105.4
AN     V3201.1
OLD
LD     V105.5
AN     V3201.4
OLD
LD     V105.6
AN     V3201.7
OLD
LD     V105.7
AN     V3202.2
OLD
LD     V17.4
AN     V3202.5
OLD
O      V3400.0
TON    T189, +20
=      M1.2
Network 189
LD     V105.1
A      V3200.1
LD     V105.2
A      V3200.4
OLD
LD     V105.3
A      V3200.7
OLD
LD     V105.4
A      V3201.2
OLD
LD     V105.5
A      V3201.5
OLD
LD     V105.6
A      V3202.0
OLD
LD     V105.7
A      V3202.3
OLD
LD     V17.4
A      V3202.6
OLD
=      V3400.0
Network 190
LD     M10.0
EU
S      M26.0, 1
Network 191
LD     M26.0
A      SM0.5
EU
LD     SM0.1
LD     T156
A      M11.1
OLD
O      M27.0
O      M26.5
EU
CTU    C0, +0
Network 192
LD     M11.1
TON    T156, +1
Network 193
LD     M11.1
EU
MOVW   C0, VW1200
Network 194
LD     M11.1
A      T156
O      SM0.1
O      M27.0
O      M26.5
R      M26.0, 1
Network 195
LD     M11.1
AN     C2
EU
LD     SM0.1
O      M26.5
CTU    C2, +2
Network 196
LD     C2
EU
MOVW   VW1200, VW1204
Network 197
LD     M12.0
EU
S      M26.1, 1
Network 198
LD     M13.1
A      T155
O      SM0.1
O      M26.5
O      M27.0
R      M26.1, 1
Network 199
LD     M26.1
A      SM0.5
EU
LD     T155
A      M13.1
O      SM0.1
O      M27.0
O      M26.5
CTU    C3, +0
Network 200
LD     M13.1
TON    T155, +1
Network 201
LD     M13.1
EU
MOVW   C3, VW1300
Network 202
LD     M13.1
AN     C5
EU
LD     SM0.1
O      M26.5
CTU    C5, +2
Network 203
LD     C5
EU
MOVW   VW1300, VW1304
Network 204
LD     C2
A      C5
AW>=   VW1304, VW1204
MOVW   VW1304, VW1308
Network 205
LD     C2
A      C5
AW<    VW1304, VW1204
MOVW   VW1204, VW1308
Network 206
LD     C2
A      C5
MOVW   VW1308, VW1320
*I     +10, VW1320
Network 207
LD     C2
A      C5
MOVW   VW1320, VW1318
+I     +0, VW1318
Network 208
LD     C2
A      C5
MOVW   VW1318, VW1310
/I     +2, VW1310
Network 209
LD     C2
A      C5
MOVW   VW1310, VW1316
*I     +10, VW1316
Network 210
LD     SM0.0
MOVW   VW3800, VW3802
*I     +10, VW3802
Network 211
LD     SM0.0
MOVW   VW3802, VW3804
+I     +30, VW3804
Network 212
LD     M26.5
EU
MOVW   VW3804, VW1316
Network 213
LD     M26.5
O      SM0.1
LPS
MOVW   +0, VW1204
AENO
MOVW   +0, VW1320
LPP
MOVW   +0, VW1304
Network 214
LD     M26.5
O      SM0.1
LPS
MOVW   +0, VW1310
AENO
MOVW   +0, VW1312
AENO
MOVW   +0, VW1314
LPP
MOVW   +0, VW1200
AENO
MOVW   +0, VW1300
Network 215
LD     M0.0
AN     C2
MOVW   VW2072, VW4524
Network 216
LDW<>  VW2072, VW4524
=      M26.5
Network 217
LD     M0.0
MOVW   VW204, VW2070
+I     VW210, VW2070
Network 218
LD     M0.0
MOVW   VW2070, VW2072
+I     VW216, VW2072
Network 219
LD     V104.1
O      SM0.1
R      M10.0, 16
R      M12.0, 16
END_SUBROUTINE_BLOCK
